(* CoDeSys 2.3 export: CLOCK01S.EXP *)

(* POU clock01s, ST *)
PROGRAM clock01s
VAR
END_VAR
clock01secImpulse:=1;
END_PROGRAM
